FUNCTION_BLOCK PUBLIC EventEmitterInterface_TestSuite EXTENDS TcUnit.FB_TestSuite
VAR
END_VAR

CheckEmitWorksWithHandler();
CheckExtendsFromQueryInterface();
CheckOffEventUnregistersAHandler();
CheckOnceEventCorrectlyCallsHandler();

METHOD PUBLIC CheckEmitWorksWithHandler
VAR
	mockEvent : MockEvent;
	mockHandler : MockEventHandler;
	eventEmitter : EventEmitter;
	iEventEmitter : I_EventEmitter := eventEmitter;
	eventReceived : BOOL;
END_VAR
TEST('CheckEmitWorksWithHandler');

iEventEmitter.OnEvent('test', mockHandler);

eventEmitter.Emit('test',mockEvent);
eventReceived := mockHandler.EqualsLastEvent(mockEvent);

AssertTrue(
	Condition := eventReceived,
	Message := 'Event Emitter did not correctly emmit the event to the handler'
);

TEST_FINISHED();
END_METHOD

METHOD PUBLIC CheckExtendsFromQueryInterface
VAR
	eventEmitter : EventEmitter;
	iEventEmitter : I_EventEmitter := eventEmitter;
	iQueryInterface : __SYSTEM.IQueryInterface;
	result : BOOL;
END_VAR
TEST('CheckExtendsFromQueryInterface');

result := __QUERYINTERFACE(iEventEmitter,iQueryInterface);

AssertTrue(
	Condition := result,
	Message := 'Interface did not extend __SYSTEM.IQueryInterface'
);

TEST_FINISHED();
END_METHOD

METHOD PUBLIC CheckOffEventUnregistersAHandler
VAR
	mockEvent : MockEvent;
	mockHandler : MockEventHandler;
	eventEmitter : EventEmitter;
	iEventEmitter : I_EventEmitter := eventEmitter;
	eventReceived : BOOL;
END_VAR
TEST('CheckOffEventUnregistersAHandler');

iEventEmitter.OnEvent('test', mockHandler);
iEventEmitter.OffEvent('test', mockHandler);

eventEmitter.Emit('test',mockEvent);
eventReceived := mockHandler.EqualsLastEvent(mockEvent);

AssertFalse(
	Condition := eventReceived,
	Message := 'Event Emitter did not correctly unregister the event handler using the off method'
);

TEST_FINISHED();
END_METHOD

METHOD PUBLIC CheckOnceEventCorrectlyCallsHandler
VAR
	mockEvent : MockEvent;
	mockHandler : MockEventHandler;
	eventEmitter : EventEmitter;
	iEventEmitter : I_EventEmitter := eventEmitter;
	eventReceived : BOOL;
END_VAR
TEST('CheckOnceEventCorrectlyCallsHandler');

iEventEmitter.OnceEvent('test', mockHandler);

eventEmitter.Emit('test',mockEvent);
eventReceived := mockHandler.EqualsLastEvent(mockEvent);

AssertTrue(
	Condition := eventReceived,
	Message := 'Event Emitter did not notify the handler'
);

TEST_FINISHED();
END_METHOD

END_FUNCTION_BLOCK

(* stored: Version 1.1.0.1, ProductVersion 3.1.4024.12
   POU EventEmitterInterface_TestSuite: Id {8094199c-ac7c-010f-03fb-a580bad4071e}, SpecialFunc None
   Method CheckEmitWorksWithHandler: Id {62729e64-7ce6-0303-1e2d-9356c48cd1f0}
   Method CheckExtendsFromQueryInterface: Id {10b34bbe-f70e-00d9-14a3-badcdd435489}
   Method CheckOffEventUnregistersAHandler: Id {9556df52-5439-0aa7-00a4-c80f384af142}
   Method CheckOnceEventCorrectlyCallsHandler: Id {4a021e24-4acc-0499-2258-14a7364b42c7} *)
